// TIA Portal V20 export
FUNCTION_BLOCK "CallEquipmentMotionCycle"   // FB209, LAD
// stored: IsIECCheckEnabled true, MemoryReserve 100, Namespace Unit1.Em0, SetENOAutomatically true
   VAR_INPUT
      diameter : LReal;
      dancer : LReal;
   END_VAR
   VAR_OUTPUT
      error { ExternalAccessible := 'False'; ExternalVisible := 'False'; ExternalWritable := 'False'} : Bool;
   END_VAR
   VAR_IN_OUT
      syncNode : "Unit1.Em0.typeSyncNode";
      axis : Array[1.._.U1EM0_NO_OF_AXES] of DB_ANY;
   END_VAR
   VAR
      instSequenceUnwinderCycle : "Unit1.Em0.SequenceUnwinderCycle";
   END_VAR
   VAR_TEMP
      tempSyncNodes : "Unit1.Em0.typeSyncNode";
   END_VAR
BEGIN

REGION Network 1 (SCL): Copy sync node inputs to temp
   #tempSyncNodes.commands := #syncNode.commands;
END_REGION

REGION Network 2: Call Sequence
   // Add logic here, that should be executed in the Motion cycle. This logic called in OB MC_PreInterpolator. This could be e.g. immediate positioning commands.
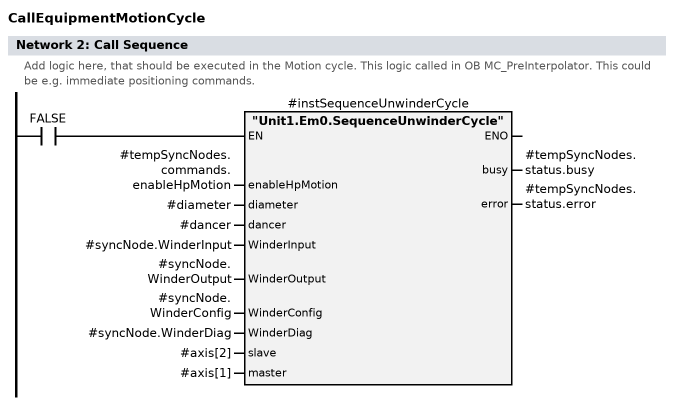
   RUNG wire#powerrail
      Contact( FALSE )
      #instSequenceUnwinderCycle(enableHpMotion := #tempSyncNodes.commands.enableHpMotion, diameter := #diameter, dancer := #dancer, WinderInput := #syncNode.WinderInput, WinderOutput := #syncNode.WinderOutput, WinderConfig := #syncNode.WinderConfig, WinderDiag := #syncNode.WinderDiag, slave := #axis[2], master := #axis[1], busy => #tempSyncNodes.status.busy, error => #tempSyncNodes.status.error)
   END_RUNG
   // the same network as SCL:
   IF FALSE THEN
       #instSequenceUnwinderCycle(enableHpMotion := #tempSyncNodes.commands.enableHpMotion,   // "Unit1.Em0.SequenceUnwinderCycle"
                               diameter := #diameter,
                               dancer := #dancer,
                               WinderInput := #syncNode.WinderInput,
                               WinderOutput := #syncNode.WinderOutput,
                               WinderConfig := #syncNode.WinderConfig,
                               WinderDiag := #syncNode.WinderDiag,
                               slave := #axis[2],
                               master := #axis[1],
                               busy => #tempSyncNodes.status.busy,
                               error => #tempSyncNodes.status.error);
   END_IF;
END_REGION

REGION Network 3 (SCL): Copy sync node outputs from temp
   #syncNode.status := #tempSyncNodes.status;
END_REGION
END_FUNCTION_BLOCK
